FUNCTION_BLOCK FB_RCC
VAR_IN_OUT
	stRCC_VRC_01 : ST_VRC;
	stRCC_VRC_02 : ST_VRC;
	stRCC_VRC_03 : ST_VRC;
	stRCC_VRC_04 : ST_VRC;
	stRCC_GCP_01 : ST_VG;
END_VAR
VAR
	{attribute 'pytmc' :=' pv: ILK_Setpoint '}
    RCC_GCP_01_INTERLOCK_SETPOINT : REAL := 10;
	{attribute 'pytmc' :=' pv: OverrideMode '}
	xSystemOverrideMode_RCC : BOOL := FALSE;
	{attribute 'pytmc' :=' pv: sLogMessage '}
	sLogMessage : T_MaxString := '';
	
	T1 : TIME := T#20s;
	T2 : TIME := T#10s;
	T3 : TIME := T#5s;
	T4 : TIME := T#10s;
	RUN_CLEAN : BOOL := TRUE;
	
	fbFormat   : FB_FormatString;
	
	tTimer1 : TON;
	current_state : INT := -1;
	init_cycle : BOOL  := FALSE;
	
	RCC_VRC_01_OPEN_OK : BOOL;
    RCC_VRC_02_OPEN_OK : BOOL;
    RCC_VRC_03_OPEN_OK : BOOL;
    RCC_VRC_04_OPEN_OK : BOOL;
END_VAR


(* Valve can open only when CRIX-RCC-VRC-02 and 03 are closed*)
RCC_VRC_01_OPEN_OK := ( stRCC_VRC_02.i_xClsLS AND NOT stRCC_VRC_02.q_xOPN_DO ) AND
                                    ( stRCC_VRC_03.i_xClsLS AND NOT stRCC_VRC_03.q_xOPN_DO ) ;

(* Valve can open only when CRIX-RCC-VRC-01 and 04 are closed*)
RCC_VRC_02_OPEN_OK := ( stRCC_VRC_01.i_xClsLS AND NOT stRCC_VRC_01.q_xOPN_DO ) AND
                                    ( stRCC_VRC_04.i_xClsLS AND NOT stRCC_VRC_04.q_xOPN_DO );

(* Valve can open only when CRIX-RCC-GCP-01 reading < setpoint Torr and CRIX-RCC-VRC-01 and 04 are closed*)
RCC_VRC_03_OPEN_OK := (stRCC_GCP_01.rPRESS < RCC_GCP_01_INTERLOCK_SETPOINT AND stRCC_GCP_01.xPRESS_OK ) AND
                                 ( stRCC_VRC_01.i_xClsLS AND NOT stRCC_VRC_01.q_xOPN_DO ) AND
                                              ( stRCC_VRC_04.i_xClsLS AND NOT stRCC_VRC_04.q_xOPN_DO );


(* Valve can open only when CRIX-RCC-VRC-02 and 03 are closed*)
RCC_VRC_04_OPEN_OK := ( stRCC_VRC_02.i_xClsLS AND NOT stRCC_VRC_02.q_xOPN_DO ) AND
                                      ( stRCC_VRC_03.i_xClsLS AND NOT stRCC_VRC_03.q_xOPN_DO ) ;
			
 CASE current_state OF
	-1:
		IF init_cycle THEN 
			current_state := 0; 
			init_cycle := FALSE;
		END_IF
		
	0:
		stRCC_VRC_01.q_xOPN_DO := FALSE;
		stRCC_VRC_02.q_xOPN_DO := FALSE;
		stRCC_VRC_03.q_xOPN_DO := FALSE;
		stRCC_VRC_04.q_xOPN_DO := FALSE;
		current_state:=1;
		
	1: // OPEN
		tTimer1(IN:=TRUE, PT:=T1);
		stRCC_VRC_02.q_xOPN_DO := TRUE;
	
		IF tTimer1.Q THEN 
			current_state := 2;
			tTimer1(IN:=FALSE); // RESTART TIMER
		END_IF
		
	2:	// DRAIN_1
		// THIS MIGHT CAUSE THE RCC TO STALL IF THIS CONDITION IS NEVER MET
		IF RCC_VRC_03_OPEN_OK THEN
			IF run_clean THEN stRCC_VRC_02.q_xOPN_DO := FALSE; END_IF
			stRCC_VRC_03.q_xOPN_DO := TRUE;
			current_state := 3; 
		END_IF
		
	3:	// DRAIN_2
		tTimer1(IN:=TRUE, PT:=T2);
		
		IF tTimer1.Q THEN 
			current_state := 4;
			IF NOT RCC_VRC_03_OPEN_OK THEN current_state := 1; END_IF
 			stRCC_VRC_03.q_xOPN_DO := FALSE;
			IF NOT run_clean THEN stRCC_VRC_02.q_xOPN_DO := FALSE; END_IF
			tTimer1(IN:=FALSE); // RESTART TIMER
		END_IF
		
	4: // OPEN VRC_01 for T3
		tTimer1(IN:=TRUE, PT:=T3);
		stRCC_VRC_01.q_xOPN_DO := TRUE;
		IF tTimer1.Q THEN 
			current_state := 5;
			tTimer1(IN:=FALSE); // RESTART TIMER
		END_IF
		
	5: // OPEN VRC_04 for T4
		tTimer1(IN:=TRUE, PT:=T4);
		stRCC_VRC_04.q_xOPN_DO := TRUE;
		IF tTimer1.Q THEN 
			current_state := -1;
			stRCC_VRC_01.q_xOPN_DO := FALSE;
			stRCC_VRC_04.q_xOPN_DO := FALSE;
			tTimer1(IN:=FALSE); // RESTART TIMER
		END_IF	
	
	
END_CASE

METHOD start_cycle : BOOL
VAR_INPUT
END_VAR
start_cycle := init_cycle := TRUE;
END_METHOD

END_FUNCTION_BLOCK

(* stored: Version 1.1.0.1, ProductVersion 3.1.4024.15
   POU FB_RCC: Id {47a0acf2-060b-4e55-9edc-089d8f8e62bc}, SpecialFunc None
   Method start_cycle: Id {0638d37b-98e4-4dcd-b1fe-fea9c7d7701d} *)
